TEXTLIST S1_Prompts
  0 = 'Station 1 Prompt'
  1 = 'prompt 2'
  2 = 'prompt 3'
   = ''
END_TEXTLIST

(* stored: Version 1.1.0.1, ProductVersion 3.1.4024.12
   TextList S1_Prompts: Id {13a16649-1219-0fa1-2fcb-27f0938a9682} *)
